# EPICS substitutions: iocBoot/iocvxWorks/canberra_13.substitutions
file "$(MCA)/mcaApp/Db/simple_mca.db"
{
pattern
{P           M       DTYP           INP         PREC  CHANS}
{CARS:med:   mca1  "asynMCA"   "@asyn(AIM2/1 0)"    3  2048}
{CARS:med:   mca2  "asynMCA"   "@asyn(AIM2/1 1)"    3  2048}
{CARS:med:   mca3  "asynMCA"   "@asyn(AIM2/1 2)"    3  2048}
{CARS:med:   mca4  "asynMCA"   "@asyn(AIM2/2 0)"    3  2048}
{CARS:med:   mca5  "asynMCA"   "@asyn(AIM2/2 1)"    3  2048}
{CARS:med:   mca6  "asynMCA"   "@asyn(AIM2/2 2)"    3  2048}
{CARS:med:   mca7  "asynMCA"   "@asyn(AIM3/1 0)"    3  2048}
{CARS:med:   mca8  "asynMCA"   "@asyn(AIM3/1 1)"    3  2048}
{CARS:med:   mca9  "asynMCA"   "@asyn(AIM3/1 2)"    3  2048}
{CARS:med:   mca10 "asynMCA"   "@asyn(AIM3/2 0)"    3  2048}
{CARS:med:   mca11 "asynMCA"   "@asyn(AIM3/3 1)"    3  2048}
{CARS:med:   mca12 "asynMCA"   "@asyn(AIM3/4 2)"    3  2048}
{CARS:med:   mca13 "asynMCA"   "@asyn(AIM3/2 3)"    3  2048}
{CARS:med:   mca0  "Soft Channel"   ""     3  2048}
}

file "$(MCA)/mcaApp/Db/icb_amp.db"
{
pattern
{P			AMP		PORT}
{CARS:med:	amp1	"icbAmp1"}
{CARS:med:	amp2	"icbAmp2"}
{CARS:med:	amp3	"icbAmp3"}
{CARS:med:	amp4	"icbAmp4"}
{CARS:med:	amp5	"icbAmp5"}
{CARS:med:	amp6	"icbAmp6"}
{CARS:med:	amp7	"icbAmp7"}
{CARS:med:	amp8	"icbAmp8"}
{CARS:med:	amp9	"icbAmp9"}
{CARS:med:	amp10	"icbAmp10"}
{CARS:med:	amp11	"icbAmp11"}
{CARS:med:	amp12	"icbAmp12"}
{CARS:med:	amp13	"icbAmp13"}
}

file "$(MCA)/mcaApp/Db/icb_adc.db"
{
pattern
{P			ADC		PORT}
{CARS:med:	adc1	"icbAdc1"}
{CARS:med:	adc2	"icbAdc2"}
{CARS:med:	adc3	"icbAdc3"}
{CARS:med:	adc4	"icbAdc4"}
}

file "$(MCA)/mcaApp/Db/icb_hvps.db"
{
pattern
{P			HVPS	LIMIT	PORT}
{CARS:med:	hvps1	1000	"icbHvps1"}
}
